Fanuc KAREL source: wcnstntpath.kl

PROGRAM wcnstntpath
%NOLOCKGROUP
VAR
  p : POSITION
  q : POSITION
  i : INTEGER
  r : REAL
BEGIN
  WITH $CNSTNT_PATH = TRUE MOVE TO p
END wcnstntpath
